// Mitsubishi GX Works2 project: BookEX5_2 Operator   PLC: Q13UDV

TYPE DateTime : STRUCT
  Year : INT;
  Month : INT;
  Day : INT;
  WeekDay : INT;
  iHour : INT;
  iMin : INT;
  iSec : INT;
  ms : INT;
END_STRUCT END_TYPE

TYPE Vector : STRUCT
  axisX : REAL;
  axisY : REAL;
  axisZ : REAL;
END_STRUCT END_TYPE

TYPE WordBit : STRUCT
  Data : DWORD;
  Flag : BOOL;
END_STRUCT END_TYPE

// global labels: Global
VAR_GLOBAL
  bVar0 AT M5000 : BOOL;
  abArray0 AT M5010 : ARRAY [0..49] OF BOOL;
  sStr0 AT D5000 : STRING[199];
  sStr1 AT D5100 : STRING[199];
  sStr2 AT D5200 : STRING[199];
  sStr3 AT D5300 : STRING[199];
  sStr4 AT D5400 : STRING[199];
  sStr5 AT D5500 : STRING[199];
  sStr6 AT D5600 : STRING[199];
  sStr7 AT D5700 : STRING[199];
  sStr8 AT D5800 : STRING[199];
  sStr9 AT D5900 : STRING[199];
  iVar0 AT D4500 : INT;
  iVar1 AT D4501 : INT;
  iVar2 AT D4502 : INT;
  iVar3 AT D4503 : INT;
  iVar4 AT D4504 : INT;
  iVar5 AT D4505 : INT;
  iVar6 AT D4506 : INT;
  iVar7 AT D4507 : INT;
  iVar8 AT D4508 : INT;
  iVar9 AT D4509 : INT;
  dVar0 AT D4510 : DINT;
  dVar1 AT D4512 : DINT;
  dVar2 AT D4514 : DINT;
  dVar3 AT D4516 : DINT;
  dVar4 AT D4518 : DINT;
  dVar5 AT D4520 : DINT;
  dVar6 AT D4522 : DINT;
  dVar7 AT D4524 : DINT;
  dVar8 AT D4526 : DINT;
  dVar9 AT D4528 : DINT;
  wVar0 AT D4530 : WORD;
  wVar1 AT D4531 : WORD;
  wVar2 AT D4532 : WORD;
  wVar3 AT D4533 : WORD;
  wVar4 AT D4534 : WORD;
  wVar5 AT D4535 : WORD;
  wVar6 AT D4536 : WORD;
  wVar7 AT D4537 : WORD;
  wVar8 AT D4538 : WORD;
  wVar9 AT D4539 : WORD;
  dwVar0 AT D4540 : DWORD;
  dwVar1 AT D4542 : DWORD;
  dwVar2 AT D4544 : DWORD;
  dwVar3 AT D4546 : DWORD;
  dwVar4 AT D4548 : DWORD;
  dwVar5 AT D4550 : DWORD;
  dwVar6 AT D4552 : DWORD;
  dwVar7 AT D4554 : DWORD;
  dwVar8 AT D4556 : DWORD;
  dwVar9 AT D4558 : DWORD;
  fsVar0 AT D4560 : REAL;
  fsVar1 AT D4562 : REAL;
  fsVar2 AT D4564 : REAL;
  fsVar3 AT D4566 : REAL;
  fsVar4 AT D4568 : REAL;
  fsVar5 AT D4570 : REAL;
  fsVar6 AT D4572 : REAL;
  fsVar7 AT D4574 : REAL;
  fsVar8 AT D4576 : REAL;
  fsVar9 AT D4578 : REAL;
  fdVar0 AT D4580 : LREAL;
  tTime0 AT D4620 : TIME;
  tTime1 AT D4622 : TIME;
  tTime2 AT D4624 : TIME;
  tTime3 AT D4626 : TIME;
  tTime4 AT D4628 : TIME;
  tTime5 AT D4630 : TIME;
  tTime6 AT D4632 : TIME;
  tTime7 AT D4634 : TIME;
  tTime8 AT D4636 : TIME;
  tTime9 AT D4638 : TIME;
  tTime10 AT D4640 : TIME;
  bVar1 AT M5001 : BOOL;
  bVar2 AT M5002 : BOOL;
  bVar3 AT M5003 : BOOL;
  bVar4 AT M5004 : BOOL;
  bVar5 AT M5005 : BOOL;
  bVar6 AT M5006 : BOOL;
  bVar7 AT M5007 : BOOL;
  bVar8 AT M5008 : BOOL;
  bVar9 AT M5009 : BOOL;
  abArray1 AT M5060 : ARRAY [0..49] OF BOOL;
  abArray2 AT M5110 : ARRAY [0..49] OF BOOL;
  abArray3 AT M5160 : ARRAY [0..49] OF BOOL;
  abArray4 AT M5210 : ARRAY [0..49] OF BOOL;
  abArray5 AT M5260 : ARRAY [0..49] OF BOOL;
  abArray6 AT M5310 : ARRAY [0..49] OF BOOL;
  abArray7 AT M5360 : ARRAY [0..49] OF BOOL;
  abArray8 AT M5410 : ARRAY [0..49] OF BOOL;
  abArray9 AT M5460 : ARRAY [0..49] OF BOOL;
  fdVar1 AT D4584 : LREAL;
  fdVar2 AT D4588 : LREAL;
  fdVar3 AT D4592 : LREAL;
  fdVar4 AT D4596 : LREAL;
  fdVar5 AT D4600 : LREAL;
  fdVar6 AT D4604 : LREAL;
  fdVar7 AT D4608 : LREAL;
  fdVar8 AT D4612 : LREAL;
  fdVar9 AT D4616 : LREAL;
  aSendData1 AT D100 : ARRAY [0..9] OF INT;
  aRecvData1 AT D110 : ARRAY [0..9] OF INT;
  aSendData2 AT D120 : ARRAY [0..9] OF INT;
  aRecvData2 AT D130 : ARRAY [0..9] OF INT;
END_VAR
// user libraries (not included): HMI

FUNCTION_BLOCK AllFB
VAR_INPUT
  b_IN1 : BOOL;
  b_IN2 : BOOL;
END_VAR
VAR_OUTPUT
  b_OT : BOOL;
END_VAR
(* structured ladder/FBD written out as ST: instructions are called as NAME(EN, inputs, outputs); _pN, _eN, _tN stand for wires *)
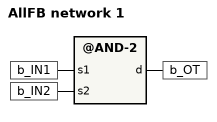
(* network 1 *)
b_OT := @AND-2(b_IN1, b_IN2);
END_FUNCTION_BLOCK

FUNCTION_BLOCK EnFB
VAR_INPUT
  b_IN1 : BOOL;
  b_IN2 : BOOL;
END_VAR
VAR_OUTPUT
  b_OT : BOOL;
END_VAR
(* structured ladder/FBD written out as ST: instructions are called as NAME(EN, inputs, outputs); _pN, _eN, _tN stand for wires *)
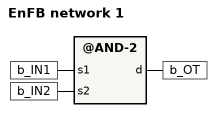
(* network 1 *)
b_OT := @AND-2(b_IN1, b_IN2);
END_FUNCTION_BLOCK

FUNCTION EnFUN
VAR_INPUT
  b_IN1 : BOOL;
  b_IN2 : BOOL;
END_VAR
(* structured ladder/FBD written out as ST: instructions are called as NAME(EN, inputs, outputs); _pN, _eN, _tN stand for wires *)
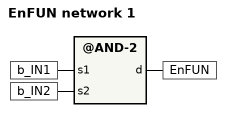
(* network 1 *)
EnFUN := @AND-2(b_IN1, b_IN2);
END_FUNCTION

FUNCTION_BLOCK MacroEnFB
VAR_INPUT
  b_IN1 : BOOL;
  b_IN2 : BOOL;
END_VAR
VAR_OUTPUT
  b_OT : BOOL;
END_VAR
(* structured ladder/FBD written out as ST: instructions are called as NAME(EN, inputs, outputs); _pN, _eN, _tN stand for wires *)
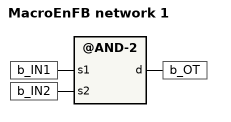
(* network 1 *)
b_OT := @AND-2(b_IN1, b_IN2);
END_FUNCTION_BLOCK

FUNCTION_BLOCK MacroFB
VAR_INPUT
  b_IN1 : BOOL;
  b_IN2 : BOOL;
END_VAR
VAR_OUTPUT
  b_OT : BOOL;
END_VAR
VAR
  ix : INT;
END_VAR
(* structured ladder/FBD written out as ST: instructions are called as NAME(EN, inputs, outputs); _pN, _eN, _tN stand for wires *)
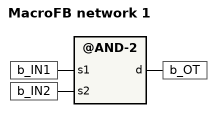
(* network 1 *)
b_OT := @AND-2(b_IN1, b_IN2);
END_FUNCTION_BLOCK

FUNCTION_BLOCK ManEnFB
VAR_INPUT
  b_EN : BOOL;
  b_IN2 : BOOL;
END_VAR
VAR_OUTPUT
  b_OT : BOOL;
END_VAR
VAR
  ix : INT;
END_VAR
VAR_INPUT
  b_IN1 : BOOL;
END_VAR
VAR_OUTPUT
  b_ENO : BOOL;
END_VAR
(* structured ladder/FBD written out as ST: instructions are called as NAME(EN, inputs, outputs); _pN, _eN, _tN stand for wires *)
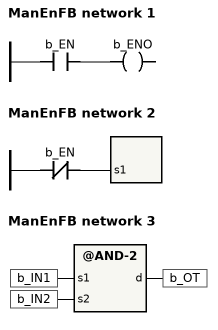
(* network 1 *)
b_ENO := b_EN;
(* network 2 *)
(* element kind 10  <- NOT b_EN *)
(* network 3 *)
b_OT := @AND-2(b_IN1, b_IN2);
END_FUNCTION_BLOCK

FUNCTION_BLOCK NoneFB
VAR_INPUT
  b_IN1 : BOOL;
  b_IN2 : BOOL;
END_VAR
VAR_OUTPUT
  b_OT : BOOL;
END_VAR
(* structured ladder/FBD written out as ST: instructions are called as NAME(EN, inputs, outputs); _pN, _eN, _tN stand for wires *)
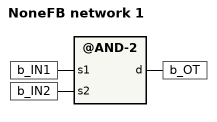
(* network 1 *)
b_OT := @AND-2(b_IN1, b_IN2);
END_FUNCTION_BLOCK

FUNCTION NoneFUN
VAR_INPUT
  b_IN1 : BOOL;
  b_IN2 : BOOL;
END_VAR
(* structured ladder/FBD written out as ST: instructions are called as NAME(EN, inputs, outputs); _pN, _eN, _tN stand for wires *)
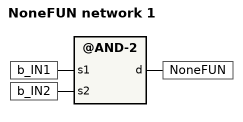
(* network 1 *)
NoneFUN := @AND-2(b_IN1, b_IN2);
END_FUNCTION

PROGRAM ExOperator
;
(*기본 연산자*)
iVar0 := iVar1 * iVar2 + iVar3 MOD 16;							(* INT *)
iVar4 := (iVar5 + D0 + iVar6) / 3;
(* iVar0 := dVar1 * iVar2 + iVar3 MOD 16;  데이터형이 틀리면 에러 *)

D0 := iVar1 * D2 + iVar3 MOD 16;
D0 := D1 * (D2+3) / 100;
(* D0 := dVar1 * dVar2 + dVar3 MOD 16;   D0는 INT로 처리함으로 에러 *)

dVar0 := dVar1 * dVar2 / 4 + dVar3 MOD 16;					(* DINT *)
dVar4 := dVar5 / H1000;
(*wVar0 := wVar1 * wVar2 + wVar3 MOD 16;  Bit-string은 일반 연산자 사용시 에러 *)

fsVar0 := fsVar1 + fsVar3 * 2.0;												(* REAL *)
fsVar1 := 2.0  * 3.14 * fsVar5;
fdVar0 := fdVar1 + fdVar2 ** 2.0;

(* sStr0 := sStr0 + "ABC";							String은 일반 연산자 사용시 에러 *)
tTime0 := tTime1+tTime2;															(* Time *)
tTime3 := tTime4 + T#1s;

(*고급 연산자*)
iVar0 := ABS(iVar2 - iVar3);														(* INT *)
dVar0 := ABS(dVar2 - dVar3);													(* DINT *)

fsVar0 := ABS(fsVar1 - fsVar2) + INT_TO_REAL(iVar0);	(* REAL *)
bVar0 := SIN_E (TRUE, fdVar1, fdVar0);
fdVar2 := SQRT((fdVar0 ** 2.0) + (fdVar1 ** 2.0));

(*논리 연산자 *)
bVar0 := bVar1 XOR M0 AND (iVar0 = 100);								(* Bit *)
D1.3 := NOT ( bVar3 AND bVar4);

D0 := D1 AND D2;																				(* WORD *)
wVar1 := wVar1 XOR wVar2;
wVar3 := wVar4 OR H0011;
D3 := D2 OR wVar1;
(* D3 := D2 OR iVar1;  D0는 WORD로  처리함으로 에러 *)

dwVar1 := dwVar1 XOR dwVar2;													(* DWORD *)
dwVar3 := NOT (dwVar4 OR dwVar1) AND H0F0F0F0F;
(* D3 := D2 OR dwVar1;  D0는 WORD로  처리함으로 에러 *)

(*관계연산자*)
bVar0 := bVar1 < bVar2;																	(* Bit *)
bVar0 := ( D0 > 100 ) AND (D0 < 200);											(* INT *)
bVar3 := dVar1 >= 100;																	(* DINT *)
bVar4 := (wVar0 AND H00FF) = 0;												(* WORD *)
bVar4 := wVar1 = H0100;
bVar4 := wVar2 > H0100;
bVar5 := (dwVar0 AND H00FF) <> 0;											(* DWORD *)
bVar6 := dwVar1 <> HFFFFFFFF;
IF D0 = 100 THEN bVar1 := TRUE; ELSE bVar1 := FALSE; END_IF;
bVar7 := tTime0 < tTime1;																(* Time *)
bVar7 := tTime2 > T#200s;
END_PROGRAM

PROGRAM 관계BIT
VAR
  bTmp1 : BOOL;
  bTmp2 : BOOL;
  bTmp3 : BOOL;
  bTmp4 : BOOL;
  bTmp5 : BOOL;
  bTmp6 : BOOL;
  bTmp7 : BOOL;
  bTmp8 : BOOL;
  bTmp9 : BOOL;
END_VAR

bTmp1 	:= TRUE;			M100 := TRUE;
bTmp2 	:= FALSE;			M101 := FALSE;
bTmp3 	:= TRUE;			D100.0 := TRUE;
bTmp4 	:= FALSE;			D100.1 := FALSE;

bVar0 := bTmp1 < bTmp2;									 
bVar1 := bTmp1 > bTmp2;		
bVar2 := bTmp1 = bTmp2;
bVar3 := bTmp1 <> bTmp2;
bVar4 := bTmp1 = bTmp3;
bVar5 := bTmp1 <> TRUE;
bVar6 := bTmp1 <> FALSE;
bVar7 := M100 = M101;
bVar8 := D100.0 <> D100.1;

IF bTmp1 > 	  bTmp2 	THEN	bTmp5 := TRUE; ELSE bTmp5 := FALSE; END_IF; 
IF bTmp1 <= bTmp2 	THEN	bTmp6 := TRUE; ELSE bTmp6 := FALSE; END_IF; 
IF bTmp1 =   bTmp2 	THEN	bTmp7 := TRUE; ELSE bTmp7 := FALSE; END_IF;  
IF bTmp1 						THEN	bTmp8 := TRUE; ELSE bTmp8 := FALSE; END_IF;  	
IF NOT bTmp2				THEN	bTmp9 := TRUE; ELSE bTmp9 := FALSE; END_IF;
END_PROGRAM

PROGRAM 관계WORD
VAR
  wTmp1 : WORD;
  bTmp1 : BOOL;
  bTmp2 : BOOL;
  bTmp3 : BOOL;
  bTmp4 : BOOL;
  bTmp5 : BOOL;
  bTmp6 : BOOL;
  bTmp7 : BOOL;
  bTmp8 : BOOL;
  bTmp9 : BOOL;
  wTmp2 : WORD;
  wTmp3 : WORD;
  wTmp4 : WORD;
  wTmp5 : WORD;
  wTmp6 : WORD;
  wTmp7 : WORD;
  wTmp8 : WORD;
  wTmp9 : WORD;
  dwTmp1 : DWORD;
  dwTmp2 : DWORD;
  dwTmp3 : DWORD;
  dwTmp4 : DWORD;
  dwTmp5 : DWORD;
  dwTmp6 : DWORD;
  dwTmp7 : DWORD;
  dwTmp8 : DWORD;
  dwTmp9 : DWORD;
END_VAR

wTmp1	:= H0055;						D100 := H0055;
wTmp2	:= H0550;						D101 := H0550;
dwTmp1	:= H00550055;					 
dwTmp2	:= H0FF00FF0;		

bVar0 := wTmp1 < wTmp2;											(* WARNING *)						 
bVar1 := WORD_TO_INT(wTmp1) > WORD_TO_INT(wTmp2);							
bVar2 := wTmp1 = wTmp2;
bVar3 := wTmp1 <> wTmp2;
bVar4 := wTmp2 = DWORD_TO_WORD(dwTmp2);
bVar5 := (wTmp1 AND wTmp3) = 0;
bVar6 := (dwTmp1 AND dwTmp2) <> 0;
bVar7 := (wTmp1 AND wTmp1) = 1;
bVar8 := wTmp1 = H0055;
bVar9 := D101 = D100;

IF wTmp1 =   wTmp2 	THEN	bTmp7 := TRUE; ELSE bTmp7 := FALSE; END_IF;  
IF dwTmp1 <> 0				THEN	bTmp8 := TRUE; ELSE bTmp8 := FALSE; END_IF;  	
IF NOT (wTmp2	<> 0)	THEN	bTmp9 := TRUE; ELSE bTmp9 := FALSE; END_IF;
END_PROGRAM

PROGRAM 관계INT
VAR
  bTmp1 : BOOL;
  bTmp2 : BOOL;
  bTmp3 : BOOL;
  bTmp4 : BOOL;
  bTmp5 : BOOL;
  bTmp6 : BOOL;
  bTmp7 : BOOL;
  bTmp8 : BOOL;
  bTmp9 : BOOL;
  iTmp1 : INT;
  iTmp2 : INT;
  iTmp3 : INT;
  iTmp4 : INT;
  iTmp5 : INT;
  iTmp6 : INT;
  iTmp7 : INT;
  iTmp8 : INT;
  iTmp9 : INT;
  dTmp1 : DINT;
  dTmp2 : DINT;
  dTmp3 : DINT;
  dTmp4 : DINT;
  dTmp5 : DINT;
  dTmp6 : DINT;
  dTmp7 : DINT;
  dTmp8 : DINT;
  dTmp9 : DINT;
  fsTmp1 : REAL;
  fsTmp2 : REAL;
  fsTmp3 : REAL;
  fsTmp4 : REAL;
  fsTmp5 : REAL;
  fsTmp6 : REAL;
  fsTmp7 : REAL;
  fsTmp8 : REAL;
  fsTmp9 : REAL;
  fdTmp1 : LREAL;
  fdTmp2 : LREAL;
  fdTmp3 : LREAL;
  fdTmp4 : LREAL;
  fdTmp5 : LREAL;
  fdTmp6 : LREAL;
  fdTmp7 : LREAL;
  fdTmp8 : LREAL;
  fdTmp9 : LREAL;
END_VAR

bTmp1		:= FALSE;						bTmp2 		:= TRUE;				D0 			:= 100;
iTmp1		:= -10;								iTmp2		:= 0; 						iTmp3 	:= 100;
dTmp1		:= -200;							dTmp2		:= 0;							dTmp3 := 200;
fsTmp1		:= -200.0;						fsTmp2		:= 0.0;						fsTmp3	:= 100.0;
fdTmp1		:= -200.0;						fdTmp2		:= 0.0;						fdTmp3	:= 100.0;
	
bVar0 := iTmp1< iTmp2;															 
bVar1 := INT_TO_DINT(iTmp2) > dTmp1;							
bVar2 := iTmp2 = REAL_TO_INT(fsTmp2);
bVar3 := fdTmp1 <> fdTmp2;
bVar4 := (ABS(iTmp3 - iTmp1) > iTmp3) AND (iTmp2 <> 0);
bVar5 := LREAL_TO_REAL(fdTmp1 * -2.0) > fsTmp3;

IF (iTmp1 < iTmp2) AND (iTmp2 < iTmp3)	THEN	bTmp5 := TRUE; ELSE bTmp5 := FALSE; END_IF;  
IF iTmp1 < iTmp2 AND iTmp2 < iTmp3			THEN	bTmp6 := TRUE; ELSE bTmp6 := FALSE; END_IF;  
IF iTmp1 < D0 						THEN	bTmp7 := TRUE; ELSE bTmp7 := FALSE; END_IF;  
IF fsTmp2 = 0.0						THEN	bTmp8 := TRUE; ELSE bTmp8 := FALSE; END_IF;  	
IF (D0 + iTmp1) > iTmp3		THEN	bTmp9 := TRUE; ELSE bTmp9 := FALSE; END_IF;
END_PROGRAM

PROGRAM 관계STR
VAR
  bTmp1 : BOOL;
  bTmp2 : BOOL;
  bTmp3 : BOOL;
  bTmp4 : BOOL;
  bTmp5 : BOOL;
  bTmp6 : BOOL;
  bTmp7 : BOOL;
  bTmp8 : BOOL;
  bTmp9 : BOOL;
END_VAR

sStr0 	:= 'ABC';			sStr1 := 'ABCD';			sStr2 := 'abcd';

bTmp1 := sStr0 < sStr1;								 
bTmp2 := sStr0 > sStr2;		
bTmp3 := sStr1 = sStr2;		 
bTmp4 := sStr2 <> sStr1;
bTmp5 := sStr1 < sStr2;
 
IF (sStr0 < sStr1) AND (sStr2 > sStr1) THEN bTmp7 := TRUE; ELSE bTmp7 := FALSE; END_IF;
IF sStr1 = 'ABCD' THEN bTmp8 := TRUE; ELSE bTmp8 := FALSE; END_IF;
IF sStr2 = 'ABCD' THEN bTmp9 := TRUE; ELSE bTmp9 := FALSE; END_IF;
END_PROGRAM

PROGRAM 관계TIME
VAR
  bTmp1 : BOOL;
  bTmp2 : BOOL;
  bTmp3 : BOOL;
  bTmp4 : BOOL;
  bTmp5 : BOOL;
  bTmp6 : BOOL;
  bTmp7 : BOOL;
  bTmp8 : BOOL;
  bTmp9 : BOOL;
END_VAR

tTime0	:= T#100s;			tTime1	:= T#200s;			tTime2	:= T#300s;
 
bTmp1 := tTime0 < tTime1;								 
bTmp2 := tTime2 > tTime1;		
bTmp3 := tTime1 = T#200s;		 
bTmp4 := tTime1 <> tTime3;
 
IF tTime1 = tTime2 		THEN bTmp8 := TRUE; ELSE bTmp8 := FALSE; END_IF;
IF tTime2 <> T#100h 	THEN bTmp9 := TRUE; ELSE bTmp9 := FALSE; END_IF;
END_PROGRAM

PROGRAM 기본
VAR
  aBoxNo : ARRAY [0..99] OF INT;
  aStr : ARRAY [0..9] OF STRING[4] := [10('')];
  aStr2 : ARRAY [0..19] OF STRING[32] := [20('')];
  ix : INT;
  Val1 : INT;
  Val2 : INT;
  Val3 : INT;
END_VAR

bVar0 	:= TRUE;			bVar1 	:= FALSE;
iVar0	:= 150;				iVar1	:= -100;
dVar0	:= 1300;			dVar1 	:= -100;
fsVar0	:= 3.0;				fsVar1	:= 4.0;
fdVar0	:= 10000.0;			fdVar1	:= 200.0;
wVar0	:= H0055;			wVar1	:= H0100;
dwVar0 	:= H0055;			dwVar1 	:= HFFFFFFFF;
tTime0	:= T#100s;			tTime1	:= T#200s;
sStr0	:= ' 12345';		sStr1	:= '-23456';
 
(* BIT *)
iVar6 	:= BOOL_TO_INT(bVar0) + BOOL_TO_INT(bVar1);									 
bVar2 	:= INT_TO_BOOL(BOOL_TO_INT(bVar0) - 1);	
bVar3 	:= INT_TO_BOOL(BOOL_TO_INT(bVar1) + 12);	
(* WORD *)	 
iVar7	:= WORD_TO_INT(wVar0) * WORD_TO_INT(wVar1);
wVar3	:= INT_TO_WORD(WORD_TO_INT(wVar0) * WORD_TO_INT(wVar1)); 
(* DWORD *)
dVar8	:= DWORD_TO_DINT(dwVar1) * 2;
dwVar3	:= DINT_TO_DWORD(DWORD_TO_DINT(dwVar0) - DWORD_TO_DINT(dwVar1)); 
(* INT *)
iVar2 	:= iVar0 + iVar1;
iVar3	:= iVar0 * (iVar0 + iVar1);
iVar4	:= iVar0 / 50 + iVar1 / 2;
(* DINT *)
dVar6	:= dVar0 + dVar1 + INT_TO_DINT(iVar0);
dVar7	:= dVar0 / dVar1;
(* Single precision*)
fsVar6	:= fsVar0**2 + fsVar1**2;
fsVar7	:= fsVar0 / fsVar1;
(* Double precision*)
fdVar6	:= 100.0 + fdVar0 * fdVar1;
fdVar7	:= fdVar0 / fdVar1 * 2.0;
(* Time *)	
tTime2	:= tTime0 + tTime1;				
tTime3	:= tTime2 - T#200s;
tTime4	:= tTime2 * 2;
(* String *)	
sStr2	:= INT_TO_STR(STR_TO_INT(sStr0) + 1);				
sStr3	:= INT_TO_STR(STR_TO_INT(sStr1) - 12);
END_PROGRAM

PROGRAM 고급
VAR
  aBoxNo : ARRAY [0..99] OF INT;
  aStr : ARRAY [0..9] OF STRING[4] := [10('')];
  aStr2 : ARRAY [0..19] OF STRING[32] := [20('')];
  ix : INT;
  Val1 : INT;
  Val2 : INT;
  Val3 : INT;
END_VAR

bVar0 	:= TRUE;			bVar1 	:= FALSE;
iVar0	:= 150;				iVar1	:= -100;
dVar0	:= 1300;			dVar1 	:= -100;
fsVar0	:= 3.0;				fsVar1	:= 4.0;
fdVar0	:= 10000.0;			fdVar1	:= 200.0;
wVar0	:= H0055;			wVar1	:= H0100;
dwVar0 	:= H0055;			dwVar1 	:= HFFFFFFFF;
tTime0	:= T#100s;			tTime1	:= T#200s;
sStr0	:= ' 12345';		sStr1	:= '-23456';
 
iVar0 := ABS(iVar2 - iVar3);							(* INT *)
dVar0 := ABS(dVar2 - dVar3);							(* DINT *)
fsVar2 := ABS(fsVar1 - fsVar0) + INT_TO_REAL(iVar0);	(* REAL *)
bVar3 := SIN_E (TRUE, fdVar1, fdVar0);
bVar4 := SQRT_E(TRUE, fsVar0, fsVar4); 
fsVar5 := SQRT(fsVar0);
END_PROGRAM

PROGRAM 논리
VAR
  aBoxNo : ARRAY [0..99] OF INT;
  aStr : ARRAY [0..9] OF STRING[4] := [10('')];
  aStr2 : ARRAY [0..19] OF STRING[32] := [20('')];
  ix : INT;
  Val1 : INT;
  Val2 : INT;
  Val3 : INT;
END_VAR

bVar0 	:= TRUE;			bVar1 	:= FALSE;
wVar0	:= H0055;			wVar1	:= H0100;
dwVar0 	:= H0055;			dwVar1 	:= HFFFFFFFF;
D1		:= H0F0F;			D2		:= HF0F0;
	 
(* BIT *)
bVar2 := bVar0 AND bVar1;						(* Bit *)
bVar3 := bVar0 OR bVar1;
bVar4 := NOT bVar1 OR bVar0;
bVar5 := NOT (bVar1 OR bVar0);								 
bVar6 := bVar1 XOR M0 AND (iVar0 = 100);	
D1.3  := NOT ( bVar3 & bVar4);

D0 	  := D1 AND D2;								(* WORD *)
wVar1 := wVar1 XOR wVar2;
wVar3 := wVar4 OR H0011;
D3    := D2 OR wVar1;
dwVar1:= dwVar1 & dwVar2;						(* DWORD *)
dwVar3:= NOT (dwVar4 OR dwVar1) AND H0F0F0F0F;
END_PROGRAM

PROGRAM ExError
VAR
  wTemp : WORD;
END_VAR
;

wVar0 	:= H8000;
wTemp	:= H1234;
bVar0 	:= (wVar0 AND 32768) = 32768;
wVar1 	:= wVar0 AND 32768;
bVar1 	:= (wVar0 AND H8000) = H8000;
wVar2 	:= wVar0 AND H8000;
bVar2 	:= (wVar0 AND 32768) = DINT_TO_WORD(32768);
END_PROGRAM

PROGRAM 대입
VAR
  v3DSrc : Vector;
  aiPos1 : ARRAY [0..3] OF INT;
  v3DDst : Vector;
  aiPos2 : ARRAY [0..3] OF INT;
END_VAR
;

v3DSrc.axisX := 10.0;
v3DSrc.axisY := 20.0;
v3DSrc.axisZ := 30.0;
v3DDst := v3DSrc;

aiPos1[0] := 0;
aiPos1[1] := 100;
aiPos1[2] := 200;
aiPos1[3] := 300;
aiPos2 := aiPos1;

fsVar0 := v3DDst .axisX + v3DDst .axisY + v3DDst .axisZ;
iVar0 := aiPos2[1] + aiPos2[2] + aiPos2[3];


FOR iVar0 := 0 TO 3 DO
	aiPos1[iVar0] := aiPos2[iVar0];
END_FOR;


FOR iVar1 := 0 TO 3 BY 2 DO		(* iVar1은 0, 2 순서로 바뀜 *)
    aiPos1[iVar1] := 0;
END_FOR;


D1 := 0;
REPEAT
	D1 := D1+1;
	UNTIL D1 > 100
END_REPEAT;
END_PROGRAM

PROGRAM CASE문
VAR CONSTANT
  cPhase1 : INT := 1;
END_VAR
VAR
  Res2 : INT;
  Res3 : INT;
END_VAR
;
CASE iVar0 OF
 	0 :	Res2 := iVar0 + 5;
	1 :	Res2 := iVar0 + 10;
	2 :	Res2 := iVar0 + 15;
	3 :	Res2 := iVar0 + 20;
	4 :	Res2 := iVar0 + 25;
    5:		Res2 := iVar0 + 30;
	ELSE
			Res2 := 0;
END_CASE;

CASE iVar0 OF
 	0,1,2 : Res3 := (iVar0+1) * 5 + iVar0;
	3..5,6   :	Res3 := (iVar0+1) * 5 + iVar0;
	ELSE
			Res3 := 0;
END_CASE;
END_PROGRAM

PROGRAM REPEAT문
;

D1 := 0;
REPEAT
	D1 := D1+1;
	UNTIL D1 > 100
END_REPEAT;
END_PROGRAM
